{attribute 'GeneratedUsingTerminal: EL7031-0000-0016'}
{attribute addProperty BoxType "EL7031-0000-0016"}
{attribute addProperty Id "AdsAddrAT %I*.TcoAmsAddr0Chn0AT %I*USINT1StateAT %I*UINT2"}
{attribute addProperty CRC "2173271299"}
{attribute addProperty Size "3"}
TYPE InfoData_81897D03 :
STRUCT
	{attribute addProperty Name "AdsAddr"}
	AdsAddr AT %I* : .TcoAmsAddr;
	{attribute addProperty Name "Chn0"}
	Chn0 AT %I* : USINT;
	{attribute addProperty Name "State"}
	State AT %I* : UINT;
END_STRUCT
END_TYPE

(* stored: Version 1.2.0.0, ProductVersion 3.1.4024.9
   DUT InfoData_81897D03: Id {957b3a68-9ae7-4631-b948-69aa5943a6e6} *)
